{attribute 'qualified_only'}

//-----------------------------------------------------------------------------------------
//
//                  				GV_Cyltronic
//
//								Variables Cyltronic 			
//-----------------------------------------------------------------------------------------
//
//Auteur: G.GOETZ
//Création: 04.03.2026
//Dernière modification : 04.03.2026 (G.GOETZ)
//       			
//-----------------------------------------------------------------------------------------
//
//     							Liste des modifications  	
//
// 04.03.2026 (G.GOETZ) -> Création		
//-----------------------------------------------------------------------------------------

VAR_GLOBAL PERSISTENT
END_VAR

VAR_GLOBAL
	
	(** ARRAY ST **)
		aId	: ARRAY[1..iMaxCyltronic] OF ST_Cyltronic ; // Cyltronic Structure
	
	(** PROCESS FLAG **)
	
	(** ST **)
		stMisc : ST_Miscellaneous ; // Miscellaneous if need
	
END_VAR

VAR_GLOBAL CONSTANT
	
	(** CONSTANT INT **)
		iMaxCyltronic : INT := 1 ; // Max Cyltronic
	
END_VAR

(* stored: Version 1.1.0.1, ProductVersion 3.1.4026.17
   GVL GV_Cyltronic: Id {92439e7f-43ae-4d45-af13-c45c42c5bc3d} *)
